FUNCTION_BLOCK CM_Sensor2State_V2
VAR_INPUT
	PI_ManualMode : BOOL;
	PI_AutoMode : BOOL;
	
	PI_HMI_HAND : BOOL;
	PI_HMI_HAND_ON : BOOL;
	
	PI_Manual_ON : BOOL;
	PI_AutoHigh : BOOL;
	
	PI_AlarmHighEnable : BOOL;
	PI_AlarmLowEnable : BOOL;
	PI_Alarmdelay_H : DINT;
	PI_Alarmdelay_L : DINT;
	
	PI_Alarm_Condition_H : BOOL;
	PI_Alarm_Condition_L : BOOL;
	
	
	
END_VAR
VAR_OUTPUT
	PO_HMI_HAND : BOOL;
	PO_Manual : BOOL;
	PO_High : BOOL;
	
	PO_Alarm_H : BOOL;
	PO_Alarm_L : BOOL;
END_VAR
VAR
	Alarm_limit_Exceeded_H : BOOL;
	Alarm_limit_Exceeded_L : BOOL;
	
	prg_scan_H : DINT; // used for alarm delay
	prg_scan_L : DINT; // used for alarm delay
	
	Alarm_Ack_H : BOOL;
	Alarm_Ack_L : BOOL;
	
	alarmDelay_H : systemTimeDelay;
	alarmDelay_L : systemTimeDelay;
	
	DelayForHistorianBit_H: TON;
	DelayForHistorianBit_L: TON;
END_VAR
VAR_IN_OUT
	CM_UDT_CTRL : Udt_CM_Sensor2State;
	Plant_control : Udt_PlantControl;
END_VAR

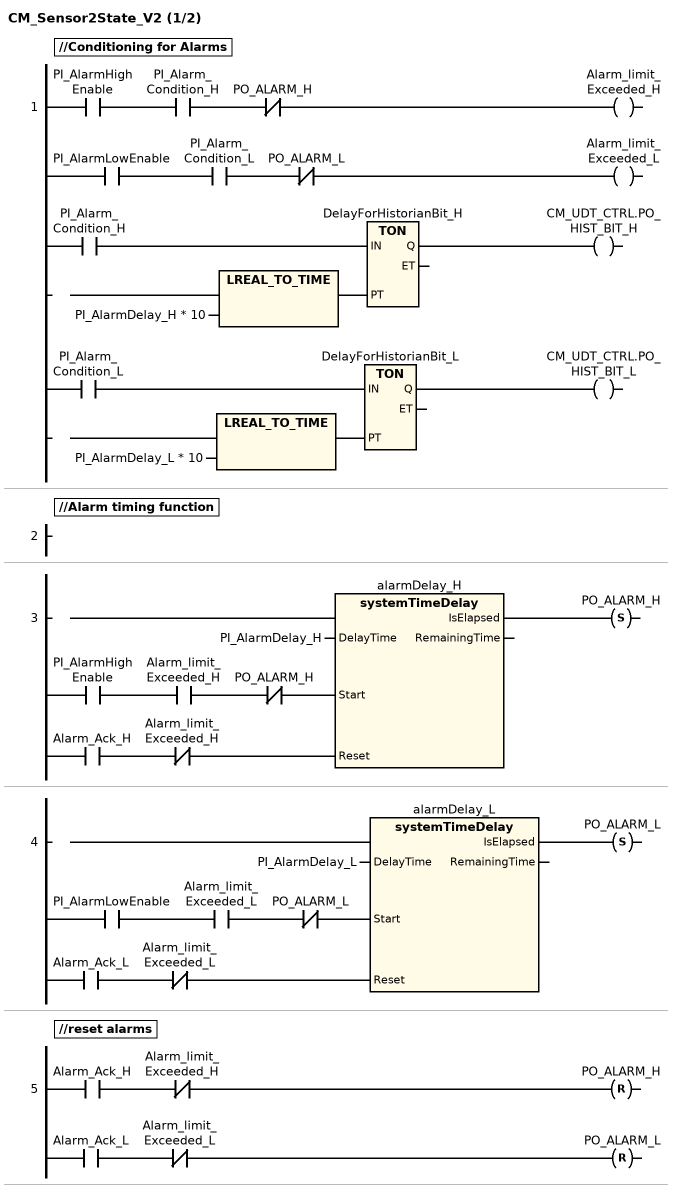
// NETWORK 1
// label: //Conditioning for Alarms
Alarm_limit_Exceeded_H := PI_AlarmHighEnable AND PI_Alarm_Condition_H AND NOT PO_ALARM_H;
Alarm_limit_Exceeded_L := PI_AlarmLowEnable AND PI_Alarm_Condition_L AND NOT PO_ALARM_L;
DelayForHistorianBit_H(IN := PI_Alarm_Condition_H, PT := LREAL_TO_TIME(PI_AlarmDelay_H * 10)); // TON
CM_UDT_CTRL.PO_HIST_BIT_H := DelayForHistorianBit_H.Q;
DelayForHistorianBit_L(IN := PI_Alarm_Condition_L, PT := LREAL_TO_TIME(PI_AlarmDelay_L * 10)); // TON
CM_UDT_CTRL.PO_HIST_BIT_L := DelayForHistorianBit_L.Q;

// NETWORK 2
// label: //Alarm timing function

// NETWORK 3
alarmDelay_H(
    DelayTime := PI_AlarmDelay_H,
    Start := PI_AlarmHighEnable AND Alarm_limit_Exceeded_H AND NOT PO_ALARM_H,
    Reset := Alarm_Ack_H AND NOT Alarm_limit_Exceeded_H); // systemTimeDelay
PO_ALARM_H S= alarmDelay_H.IsElapsed;

// NETWORK 4
alarmDelay_L(
    DelayTime := PI_AlarmDelay_L,
    Start := PI_AlarmLowEnable AND Alarm_limit_Exceeded_L AND NOT PO_ALARM_L,
    Reset := Alarm_Ack_L AND NOT Alarm_limit_Exceeded_L); // systemTimeDelay
PO_ALARM_L S= alarmDelay_L.IsElapsed;

// NETWORK 5
// label: //reset alarms
PO_ALARM_H R= Alarm_Ack_H AND NOT Alarm_limit_Exceeded_H;
PO_ALARM_L R= Alarm_Ack_L AND NOT Alarm_limit_Exceeded_L;

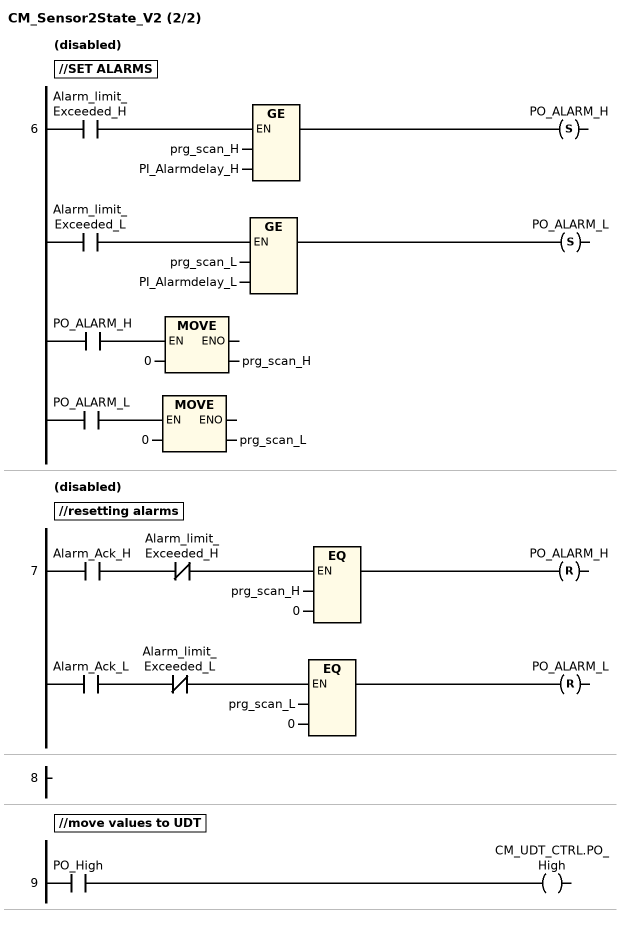
// NETWORK 6 (disabled)
// label: //SET ALARMS
// PO_ALARM_H S= Alarm_limit_Exceeded_H AND prg_scan_H >= PI_Alarmdelay_H;
// PO_ALARM_L S= Alarm_limit_Exceeded_L AND prg_scan_L >= PI_Alarmdelay_L;
// IF PO_ALARM_H THEN prg_scan_H := 0; END_IF
// IF PO_ALARM_L THEN prg_scan_L := 0; END_IF

// NETWORK 7 (disabled)
// label: //resetting alarms
// PO_ALARM_H R= Alarm_Ack_H AND NOT Alarm_limit_Exceeded_H AND prg_scan_H = 0;
// PO_ALARM_L R= Alarm_Ack_L AND NOT Alarm_limit_Exceeded_L AND prg_scan_L = 0;

// NETWORK 8

// NETWORK 9
// label: //move values to UDT
CM_UDT_CTRL.PO_High := PO_High;

END_FUNCTION_BLOCK

(* stored: Version 1.1.0.1, ProductVersion 3.1.4024.13
   POU CM_Sensor2State_V2: Id {b4ee52d5-ac68-4d40-a196-1bae48cc2784}, SpecialFunc None *)
